// TwinCAT 3 PLC project MagnetSystem_PI4
// ProgramVersion: 3.1.4023.0
// libraries:
//   CanItfHelper, * (Beckhoff Automation LLC)
//   Tc2_Math, * (Beckhoff Automation GmbH)
//   Tc2_Standard, * (Beckhoff Automation GmbH)
//   Tc2_System, * (Beckhoff Automation GmbH)
//   Tc2_TcpIp, * (Beckhoff Automation GmbH)
//   Tc2_Utilities, * (Beckhoff Automation GmbH)
//   Tc3_Module, * (Beckhoff Automation GmbH)
//   Tc3_EventLogger,3.1.30.0,Beckhoff Automation GmbH
// project tree:
//   DUTs/ E_Command.TcDUT (not stored), E_MagState.TcDUT, E_Status.TcDUT, ST_Alarm_Base.TcDUT (not stored), ST_canRxdata.TcDUT (not stored), ST_Coil_Base.TcDUT (not stored), ST_Coil_Ext_Analog1.TcDUT (not stored), ST_Control.TcDUT (not stored), ST_EngVal.TcDUT (not stored), ST_InstFeedback.TcDUT (not stored), ST_RecipeLocal.TcDUT (not stored), ST_Setpoints.TcDUT (not stored), ST_PermissivesToMainPLC.TcDUT (not stored), ST_Recipe.TcDUT (not stored), ST_SysParameters.TcDUT, ST_Trip_Base.TcDUT (not stored), ST_UC_Status.TcDUT (not stored), ST_UC_Status_Dummy.TcDUT, ST_UCDevices.TcDUT, ST_UC_Trip_Base.TcDUT (not stored)
//   GVLs/ Alarms_DB.TcGVL (not stored), Command.TcGVL (not stored), Devices.TcGVL (not stored), HMI_DB.TcGVL, Input.TcGVL, GVL.TcGVL, InstrumentReading.TcGVL, IO.TcGVL (not stored), MCP_IO.TcGVL (not stored), Output.TcGVL (not stored), Permissives_DB.TcGVL (not stored), Recipe.TcGVL (not stored), Setpoints.TcGVL, Trips_DB.TcGVL, Tx_Config.TcGVL (not stored)
//   / PlcTask.TcTTO
//   POUs/ ADC_10V.TcPOU (not stored), ADC_5V.TcPOU (not stored), Alarms.TcPOU (not stored), Alarms_FB.TcPOU (not stored), Alias.TcPOU, AnalogConversion.TcPOU (not stored), Cal_ChargeTime.TcPOU, CanInterface.TcPOU (not stored), CAN_comm_old.TcPOU (not stored), CAN_comm.TcPOU (not stored), ChargeTimeCal.TcPOU (not stored), Delay2s.TcPOU (not stored), Graphs.TcPOU (not stored), Heartbeat.TcPOU (not stored), HMI.TcPOU (not stored), MAIN.TcPOU, MODE_SELECTION_1.TcPOU (not stored), Norm_x.TcPOU, Permissives.TcPOU (not stored), ChargeRlyClose_ChargerON_Seq.TcPOU (not stored), PWMO.TcPOU (not stored), Trips.TcPOU (not stored), Tx_MasterPLC.TcPOU, VoltageOutputCal.TcPOU (not stored)

CONFIGURATION MagnetSystem_PI4
    RESOURCE PLC ON TwinCAT3
        TASK PlcTask(INTERVAL := T#10ms, PRIORITY := 20);
        PROGRAM MAIN WITH PlcTask : MAIN;
    END_RESOURCE
END_CONFIGURATION

// ---- DUTs/E_MagState.TcDUT
{attribute 'qualified_only'}
{attribute 'strict'}
TYPE E_MagState :
(
	FULL_SHUTDOWN 	:= 0,
	IDLE			:= 1, 
	READY_TO_CHARGE := 2, 
	CHARGING		:= 3, 
	CHARGE_PAUSED	:= 4,
	READY_TO_SHOOT 	:= 5, 
	SHOOTING 		:= 6, 
	POST_SHOT 		:= 7, 
	//SHUTDOWN 		:= 8, //remove
	DUMPING			:= 9,
	TRIPPED			:= 10
);
END_TYPE

// ---- DUTs/E_Status.TcDUT
{attribute 'qualified_only'}
{attribute 'strict'}
{attribute 'to_string'}
TYPE E_Status :
(
	//Actual Magnetic State
	FULL_SHUTDOWN	:= 0,
	IDLE			:= 1, 
	READY_TO_CHARGE	:= 2, 
	CHARGING		:= 3, 
	CHARGING_PAUSED := 4,		
	READY_TO_SHOOT	:= 5, 
	SHOOTING		:= 6, 
	POST_SHOT		:= 7, 
	//SHUTDOWN		:= 8, 
	DUMPING			:= 9,
	TRIPPED			:= 10,
	MANUAL_MODE		:= 11 // LOCAL MODE
) ;
END_TYPE

// ---- DUTs/ST_SysParameters.TcDUT
TYPE ST_SysParameters :
STRUCT
	NumOfCaps				: INT := 2;
	Direction				: STRING[1] :='0';
	NumOfTurns				: INT := 0;
	DriverMapping			: STRING[10] := '0';
	MaxVoltagePerCap		: INT := 0;
	MaxVoltageTotal 		: INT := 0;
	CapacitancePerCap		: INT := 88;
	TotalCapacitance		: REAL := 0.0;
	TotalCircuitResistance	: REAL := 0.0;
	//TriggerTime				: INT := 0;
END_STRUCT
END_TYPE

// ---- DUTs/ST_UC_Status_Dummy.TcDUT
TYPE ST_UC_Status_Dummy EXTENDS ST_UC_Status :
STRUCT
	R2_06_UC_Rx_cobID : UDINT;
	R2_06_UC_Rx_data : ARRAY [0..7] OF BYTE;
END_STRUCT
END_TYPE

// ---- DUTs/ST_UCDevices.TcDUT
TYPE ST_UCDevices :
STRUCT
	Status : ST_UC_Status;
END_STRUCT
END_TYPE

// ---- GVLs/HMI_DB.TcGVL
{attribute 'qualified_only'}
VAR_GLOBAL
	chargePB			: BOOL;
	shootPB				: BOOL;
	dumpPB				: BOOL;
	StartPB				: BOOL;
	StopPB				: BOOL;
	PausePB				: BOOL;			 
	RemoteModeSelected	: BOOL;
	Idle_mode			: BOOL;
	SafetyOK			: BOOL;
	AllDumpRelaysOpen	: BOOL;
	AllACInterlocksClosed : BOOL;
	AllFlybackDiodesActive	: BOOL;
	IntrumentationFaulted	: BOOL;
	AllChargesAreActive		: BOOL;
	
	ReadyToChargeRunOutTime	: DINT := 0;
	ChargingRunOutTime		: DINT := 0;
	ChargePausedRunOutTime	: DINT := 0;
	ReadyToShootRunOutTime	: DINT := 0;				
	ShootingRunOutTime		: DINT := 0;
	PostShotRunOutTime		: DINT := 0;
	DumpingRunOutTime		: DINT := 0;
	
	CoilEnable				: ARRAY [1..10] OF BOOL;
	
END_VAR

// ---- GVLs/Input.TcGVL
{attribute 'qualified_only'}
VAR_GLOBAL
//***MCP
//EL1008 - DI
	R1_01_00 AT	%I*: BOOL; //Master stop PB not pressed - black pb on mcp
	R1_01_01 AT	%I*: BOOL; //case Estop circuit okay (Rly1 (120vac)
	R1_01_02 AT %I*: BOOL; //Automatic Mode Selected (NO)
	R1_01_03 AT %I*: BOOL; //24VDC OK
	R1_01_04 AT %I*: BOOL; //spare
	R1_01_05 AT %I*: BOOL; //spare
	R1_01_06 AT %I*: BOOL; //spare
	R1_01_07 AT %I*: BOOL; //spare


//***LCP
//EL3064 - AI
	R2_01_00 		AT %I*: INT;
	R2_01_00_Status AT %I*: WORD;
	
	R2_01_01		AT %I*: INT;
	R2_01_01_Status AT %I*: WORD;
	
	R2_01_02 		AT %I*: INT;
	R2_01_02_Status AT %I*: WORD;
	
//EL1008 - DI
	R2_03_00 AT %I*: BOOL;
	R2_03_01 AT %I*: BOOL;
	R2_03_02 AT %I*: BOOL;
	R2_03_03 AT %I*: BOOL;
	R2_03_04 AT %I*: BOOL;
	R2_03_05 AT %I*: BOOL;
	R2_03_06 AT %I*: BOOL;
	R2_03_07 AT %I*: BOOL;
	
	R2_04_00 AT %I*: BOOL;
	R2_04_01 AT %I*: BOOL;
	R2_04_02 AT %I*: BOOL;
	R2_04_03 AT %I*: BOOL;
	R2_04_04 AT %I*: BOOL;
	R2_04_05 AT %I*: BOOL; //spare
	R2_04_06 AT %I*: BOOL; //spare
	R2_04_07 AT %I*: BOOL; //spare

//EL6751 - CAN Open	
	
	//R2_06_UC_Rx AT %I*		: ARRAY [0..1] OF EXTCANQUEUE; // only used for raw address.
	// each Rack has 10 caps + 1 dummy varible to park the swapped cap
	R2_06_CapNumber AT %I* : ARRAY [1..10] OF  ST_UCDevices; //only used with DBC file.
	R2_06_UC_7F_status AT %I* : ST_UC_Status_Dummy;
	
//R3****** LCP2
//EL3064 - AI
	R3_01_00 		AT %I*: INT;
	R3_01_00_Status AT %I*: WORD;
	
	R3_01_01		AT %I*: INT;
	R3_01_01_Status AT %I*: WORD;
	
	R3_01_02 		AT %I*: INT;
	R3_01_02_Status AT %I*: WORD;
	
//EL1008 - DI
	R3_03_00 AT %I*: BOOL;
	R3_03_01 AT %I*: BOOL;
	R3_03_02 AT %I*: BOOL;
	R3_03_03 AT %I*: BOOL;
	R3_03_04 AT %I*: BOOL;
	R3_03_05 AT %I*: BOOL;
	R3_03_06 AT %I*: BOOL;
	R3_03_07 AT %I*: BOOL;
	
	R3_04_00 AT %I*: BOOL;
	R3_04_01 AT %I*: BOOL;
	R3_04_02 AT %I*: BOOL;
	R3_04_03 AT %I*: BOOL;
	R3_04_04 AT %I*: BOOL;
	R3_04_05 AT %I*: BOOL; //spare
	R3_04_06 AT %I*: BOOL; //rly - output relay
	R3_04_07 AT %I*: BOOL; //spare

//EL6751 - CAN Open	
	
	//R2_06_UC_Rx AT %I*		: ARRAY [0..1] OF EXTCANQUEUE; // only used for raw address.
	// each Rack has 10 caps + 1 dummy varible to park the swapped cap
	R3_06_CapNumber AT %I* : ARRAY [1..10] OF  ST_UCDevices; //only used with DBC file.
	R3_06_UC_7F_status AT %I* : ST_UC_Status_Dummy;
	//R3_06_UC_status AT %I* : ARRAY [1..10] OF ST_UC_Status;

	//R4 
	//R5	
	//..
	//R10

END_VAR

// ---- GVLs/GVL.TcGVL
{attribute 'qualified_only'}
VAR_GLOBAL
	
	//actual_magnet_systemState	: DINT;
	error_msg					: WORD;
	shot_going_OK				: BOOL;
	shot_is_done				: BOOL;
	//RequestedMagnetSysState		: DINT;
	cap_msg						: WORD; 
	
	test						: BOOL;
	ClearAllFaults				: BOOL;
	alarm_test					: BOOL;
	
	Analog_test					: REAL;
	
	fullshutdown_to_idle        : BOOL;
	idle_to_charge				: BOOL;
	idle_to_readyToCharge		: BOOL;
	readyToCharge_to_Charging	: BOOL;
	charge_to_pause				: BOOL;
	charge_to_readyToShoot		: BOOL;
	readyToShoot_to_Shoot		: BOOL;
	shoot_to_postShot			: BOOL;
	postShot_to_shutdown		: BOOL;
	shutdown_to_idle			: BOOL;
	dump_to_idle				: BOOL;
	
	AlwaysTrue					: BOOL;
	AlwaysFalse					: BOOL;
	
	AllSystemsDischarged		: BOOL;
	AllChargerReadywithSP		: BOOL;
END_VAR

// ---- GVLs/InstrumentReading.TcGVL
{attribute 'qualified_only'}
VAR_GLOBAL
	//LCP 1 Instrument reading
	R2_01_CH00 : REAL;
	R2_01_CH01 : REAL;
	R2_01_CH02 : REAL;
	
END_VAR

// ---- GVLs/Setpoints.TcGVL
{attribute 'qualified_only'}
VAR_GLOBAL
	//HMI Input -> Setpoints -> EngVal		-> PLC ---------> Tx_Config
	//						-> SysParameters-> PLC ---------> Tx_Config
	//										   PLC - Recipe -> Tx_Config 	 
	Coil : ARRAY[1..10] OF ST_Setpoints; // EngVal & SysParameters
	
END_VAR

// ---- GVLs/Trips_DB.TcGVL
{attribute 'qualified_only'}
VAR_GLOBAL
	Coil : ARRAY[1..10] OF ST_Trip_Base;
	
	AnyEstopPressed 			: BOOL;
	SystemTripped 				: BOOL;
	InstrumentationFaulted		: BOOL;
	AnyChargeRlyFail			: BOOL;
	AnyDumpRlyFail				: BOOL;
	AnyACInterlockFail			: BOOL;
	
	AnyDCPSU_fail				: BOOL;
	AnyHVisoRelayFailed			: BOOL;
	MachineTimedOut				: BOOL;
END_VAR

// ---- POUs/MAIN.TcPOU
PROGRAM MAIN
VAR
	
	status0:BOOL;
	
END_VAR

Alias();
CAN_comm();
Tx_MasterPLC();
AnalogConversion();
Permissives();
Trips();
MODE_SELECTION_1();
Alarms();
Heartbeat();
VoltageOutputCal();
Cal_ChargeTime();


//test
//IF MCP_IO.AutoModeSelected THEN
//	Output.R2_05_07 := heartbeat.pulse_1Hz;
//END_IF

	
//sample test
IF gvl.test = TRUE THEN
	Output.R2_05_00 := TRUE;
	ELSE 
		Output.R2_05_00 := FALSE; 	
END_IF;

END_PROGRAM

// ---- POUs/Alias.TcPOU
PROGRAM Alias
VAR
	i : INT := 1; //coil 1 - 10 
	j : INT := 1;  // msg 0-1 (could be 0-31 later)
END_VAR

//R1 = MCP**
//DI
	MCP_IO.MasterStopPB_Pressed					:= Input.R1_01_00;//NC
	//MCP_IO.MasterStopPB_Pressed					:= NOT Input.R2_04_07; //Temporarily used for testing.
	MCP_IO.CageEstopCircuitOK					:= Input.R1_01_01; //NO use R2_04_07 for dev test
	MCP_IO.RemoteModeSelected					:= Input.R1_01_02; // 0 = manual, 1=auto  *temporarily used for dev test
	MCP_IO.PSU1_DCOK							:= Input.R1_01_03;
	
//R2 = Coil 1
//AI
	Devices.Coil[1].ChargeVoltageFeedback_raw 	:= Input.R2_01_00;	
	Devices.Coil[1].CurrentFeedback_raw 		:= Input.R2_01_01;
	Devices.Coil[1].Measured_Bfield_raw 		:= Input.R2_01_02;
	
//PWM O
 	Output.R2_02_00 := Devices.Coil[1].ChargerSetpoint;
	Output.R2_02_01 := Devices.Coil[1].CurrentSetpoint;


//DI
	Devices.Coil[1].PSU0_active 				:= Input.R2_03_00;
	Devices.Coil[1].Local_StopPB_Pressed 		:= NOT Input.R2_03_01; //NC 
	Devices.Coil[1].DumpRelay1_closed 			:= Input.R2_03_02;
	Devices.Coil[1].DumpRelay2_closed 			:= Input.R2_03_03;
	//Devices.Coil[1].ChargeRelay_closed 			:= Input.R2_03_04;
	Devices.Coil[1].ChargerIsEnabled 			:= Input.R2_03_05;
	//Devices.Coil[1].FlybackD1_Alive 			:= Input.R2_03_06;
	//Devices.Coil[1].FlybackD2_Alive 			:= Input.R2_03_07;
	Devices.Coil[1].PSU1_DCOK					:= Input.R2_03_06;
	Devices.Coil[1].HVisolationRelayClosed		:= Input.R2_03_07; 
	
	Devices.Coil[1].DumpResistorTemperatureHigh := Input.R2_04_00;
	Devices.Coil[1].GroundLoopCurrentDetected 	:= Input.R2_04_01;
	Devices.Coil[1].CoilTemperatureHigh 		:= Input.R2_04_02;
	Devices.Coil[1].AC_Interlock_RlyClose		:= Input.R2_04_03;  //3P contactor
	Devices.Coil[1].LossPneumaticPressure       := Input.R2_04_04;
	//Spare Input.R2_04_05;  
	Devices.Coil[1].OutputRelayOpen				:= Input.R2_04_06; // rly 5
	//Spare Input.R2_04_07;  temp used for MCP estop input
	
//DQ
	Output.R2_05_00 := Devices.Coil[1].OpenDumpRelays;
	Output.R2_05_01 := Devices.Coil[1].closeChargeRelay;
	Output.R2_05_02 := Devices.Coil[1].enableOutputToCharger;
	Output.R2_05_03 := Devices.Coil[1].CloseACInterlockRly;  //3P contactor
	Output.R2_05_04 := Devices.Coil[1].CloseHVisolationRelay; // 24VDC to control 2 120Vac HV Ross Relayas  (rly6)
	Output.R2_05_05 := Devices.Coil[1].SystemFaulted; //LCP LED AMBER
	Output.R2_05_06 := Devices.Coil[1].SystemCharging;  //LCP LED RED (charging or Charged)
	Output.R2_05_07 := Devices.Coil[1].SystemReady;  // LCP LED GREEN
	
//CANOpen
	
	//Output.R2_05_CANrequest := CAN_comm.
	Output.R2_06_CANrequest.cobId := Devices.Coil[1].CanTx_config_ID;
	Output.R2_06_CANrequest.data[0] := Devices.Coil[1].CanTx_config_request[0];
	Output.R2_06_CANrequest.data[1] := Devices.Coil[1].CanTx_config_request[1];
	Output.R2_06_CANrequest.data[2] := Devices.Coil[1].CanTx_config_request[2];
	Output.R2_06_CANrequest.data[3] := Devices.Coil[1].CanTx_config_request[3];
	Output.R2_06_CANrequest.data[4] := Devices.Coil[1].CanTx_config_request[4];
	Output.R2_06_CANrequest.data[5] := Devices.Coil[1].CanTx_config_request[5];
	Output.R2_06_CANrequest.data[6] := Devices.Coil[1].CanTx_config_request[6];
	Output.R2_06_CANrequest.data[7] := Devices.Coil[1].CanTx_config_request[7];
	
	// input
FOR i := 1 TO 10 BY 1 DO
	FOR j := 1 TO 10 BY 1 DO 
		Devices.Coil[i].UltraCap[j].Elec_AveVolt 		:= Input.R2_06_CapNumber[j].Status.Elec_AveVolt; //per cell
		Devices.Coil[i].UltraCap[j].Elec_Balancing 		:= Input.R2_06_CapNumber[j].Status.Elec_Balancing; // 0x0[Not Active], 0x1[Active], 0x2[Error], 0x3[Not Available]
		Devices.Coil[i].UltraCap[j].Elec_HighestVolt 	:= Input.R2_06_CapNumber[j].Status.Elec_HighestVolt; //per cell
		Devices.Coil[i].UltraCap[j].Elec_Imbalance 		:= Input.R2_06_CapNumber[j].Status.Elec_Imbalance;  // 0x0[No Warnings], 0x1[Warning Active], 0x2[Alarm Active], 0x3[Not Available]
		Devices.Coil[i].UltraCap[j].Elec_OverVoltage	:= Input.R2_06_CapNumber[j].Status.Elec_OverVoltage;  // 0x0[No Warnings], 0x1[Warning Active], 0x2[Alarm Active], 0x3[NOT Available] 
		Devices.Coil[i].UltraCap[j].Elec_VoltageSum		:= Input.R2_06_CapNumber[j].Status.Elec_VoltageSum; //total voltage in one UC
		Devices.Coil[i].UltraCap[j].Therm_HighestCell	:= Input.R2_06_CapNumber[j].Status.Therm_HighestCell; //C
		Devices.Coil[i].UltraCap[j].Therm_HighTemp		:= Input.R2_06_CapNumber[j].Status.Therm_HighTemp;  //0x0[No Warnings], 0x1[Warning Active], 0x2[Alarm Active], 0x3[NOT Available]
	END_FOR;
END_FOR;
	Devices.Coil[1].UltraCap_Dummy.R2_06_UC_Rx_cobID := Input.R2_06_UC_7F_status.R2_06_UC_Rx_cobID;
	Devices.Coil[1].UltraCap_Dummy.R2_06_UC_Rx_data := Input.R2_06_UC_7F_status.R2_06_UC_Rx_data;

//Recipe: Coil enable from screenroom
IF MCP_IO.RemoteModeSelected = TRUE OR HMI_DB.RemoteModeSelected = TRUE THEN
	FOR i := 1 TO 10 BY 1 DO
		Devices.Coil[i].CoilEnabled :=  Recipe.Coil[i].CoilEnable;
	END_FOR;
	
ELSIF MCP_IO.RemoteModeSelected = FALSE OR HMI_DB.RemoteModeSelected = FALSE THEN
	FOR i := 1 TO 10 BY 1 DO
		Devices.Coil[i].CoilEnabled :=  HMI_DB.CoilEnable[i];	
	END_FOR;
END_IF;


IF i > 10 THEN
	i := 1;
END_IF;

IF j > 10 THEN
	j := 1;
END_IF;

END_PROGRAM

// ---- POUs/Tx_MasterPLC.TcPOU
PROGRAM Tx_MasterPLC
VAR
	i : INT := 1;
	j : INT := 1;
	TotalCapacitance_REAL : ARRAY[1..10] OF REAL;
	
END_VAR

//Calculations for Max Total Voltage and Total Capacitance
FOR i := 1 TO 10 BY 1 DO
	Setpoints.Coil[i].SysParameters.MaxVoltageTotal := Setpoints.Coil[i].SysParameters.NumOfCaps * Setpoints.Coil[i].SysParameters.MaxVoltagePerCap;
	TotalCapacitance_REAL[i] := INT_TO_REAL(Setpoints.Coil[i].SysParameters.CapacitancePerCap) / INT_TO_REAL(Setpoints.Coil[i].SysParameters.NumOfCaps);
	Setpoints.Coil[i].SysParameters.TotalCapacitance := TotalCapacitance_REAL[i];
END_FOR


//Grouping systemParameters and configuration for sending to main plc
FOR i := 1 TO 10 BY 1 DO
	Tx_Config.CoilSP[i].SysParameters.Direction := Setpoints.Coil[i].SysParameters.Direction;
	Tx_Config.CoilSP[i].SysParameters.NumOfTurns := Setpoints.Coil[i].SysParameters.NumOfTurns;
	Tx_Config.CoilSP[i].SysParameters.DriverMapping := Setpoints.Coil[i].SysParameters.DriverMapping;
	Tx_Config.CoilSP[i].SysParameters.NumOfCaps := Setpoints.Coil[i].SysParameters.NumOfCaps;
	Tx_Config.CoilSP[i].SysParameters.MaxVoltagePerCap := Setpoints.Coil[i].SysParameters.MaxVoltagePerCap;
	Tx_Config.CoilSP[i].SysParameters.MaxVoltageTotal := Setpoints.Coil[i].SysParameters.MaxVoltageTotal;
	Tx_Config.CoilSP[i].SysParameters.CapacitancePerCap := Setpoints.Coil[i].SysParameters.CapacitancePerCap;
	Tx_Config.CoilSP[i].SysParameters.TotalCapacitance := Setpoints.Coil[i].SysParameters.TotalCapacitance;
	Tx_Config.CoilSP[i].SysParameters.TotalCircuitResistance := Setpoints.Coil[i].SysParameters.TotalCircuitResistance;
	
	Tx_Config.CoilSP[i].RecipeLocal.chargerSetpoint	:= Setpoints.Coil[i].RecipeLocal.chargerSetpoint;//calculated locally, thought the mainPLC might want to have this 
	Tx_Config.CoilSP[i].Recipe.CoilEnable			:= Recipe.Coil[i].CoilEnable;
	Tx_Config.CoilSP[i].Recipe.CurrentDuration	:= Recipe.Coil[i].CurrentDuration; //total charge time?
	Tx_Config.CoilSP[i].Recipe.currentSetpoint	:= Recipe.Coil[i].currentSetpoint;
	Tx_Config.CoilSP[i].Recipe.TriggerTime		:= Recipe.Coil[i].TriggerTime;
	
	Tx_Config.CoilInst[i].ChargerVolt := Devices.Coil[i].ChargeVoltageFeedback;
	
	FOR j := 1 TO 15 BY 1 DO 
		Tx_Config.CoilInst[i].CapVolt[j] := INT_TO_REAL (Devices.Coil[i].CapVoltage[j]); //1-15 uc
		Tx_Config.CoilInst[i].TotalVoltage := Devices.Coil[i].TotalVoltage;
	END_FOR
	
	Tx_Config.CoilInst[i].Cur := Devices.Coil[i].CurrentFeedback;
	
END_FOR

//run out time of each state
Tx_Config.ReadyToChargeRunOutTime := TIME_TO_REAL (MODE_SELECTION_1.ReadyToChargeRunOutTMR_PT);
Tx_Config.ChargingRunOutTime := TIME_TO_REAL (MODE_SELECTION_1.ChargingRunOutTMR_PT);
Tx_Config.ChargePausedRunOutTime := TIME_TO_REAL (MODE_SELECTION_1.ChargePausedRunOutTMR_PT);
Tx_Config.ReadyToShootRunOutTime := TIME_TO_REAL (MODE_SELECTION_1.ReadyToShootRunOutTMR_PT);
Tx_Config.ShootingRunOutTime := TIME_TO_REAL (MODE_SELECTION_1.ShootingRunOutTMR_PT);
Tx_Config.PostShotRunOutTime := TIME_TO_REAL (MODE_SELECTION_1.PostShotRunOutTMR_PT);
Tx_Config.DumpingRunOutTime := TIME_TO_REAL (MODE_SELECTION_1.DumpingRunOutTMR_PT);

//voltage and current feedback???

//TxRx
(*
FB_ReadAdsSymByName (
			bRead		:= TRUE, // on or off
			sNetID		:= 5.104.224.86.1.333, //AmsNetID
			nPort		:= 852, // plc port
			sVarName	:= E_Command,  //read from
			nDestAddr	:= E_Command, //write to 
			nLen		:= 2, //2 bytes	
			);

FB_WriteAdsSymByName (
			bWrite		:= TRUE,
			sNetID		:= 5.1.121.21.21.2,
			nPort		:= 851,
			sVarName	:= E_Status,
			nSrcAddr	:= E_Status,
			nLen		:= 2, //2byte
			);
*)


IF i > 10 THEN 
	i := 1;
END_IF

IF j > 15 THEN 
	j := 1;
END_IF

END_PROGRAM

// ---- POUs/Cal_ChargeTime.TcPOU
PROGRAM Cal_ChargeTime
VAR
	chargetimeCal : ARRAY [1..10] OF ChargeTimeCal;
	Tuntilfullycharged : ARRAY [1..10] OF REAL;
	i : INT := 1;
END_VAR


FOR i := 1 TO 10 BY 1 DO
	chargetimeCal[i] (I_setpoint := setpoints.Coil[i].Recipe.currentSetpoint, 
					t_duration := setpoints.Coil[i].Recipe.CurrentDuration, 
					NumOfCaps := setpoints.Coil[i].SysParameters.NumOfCaps,
					C_percap := setpoints.Coil[i].SysParameters.CapacitancePerCap,
					VMAXperCap := setpoints.Coil[i].SysParameters.MaxVoltagePerCap,
					R_coil := setpoints.Coil[i].SysParameters.TotalCircuitResistance,
					L_coil := 0.5,
					VMAXcharger := 1500,
					Pcharger := 15000,
					NumOfCharger := 4);
				
Tuntilfullycharged[i] := chargetimeCal[i].Tuntilfullcharge;
END_FOR;

IF i > 10 THEN 
	i := 1;
END_IF

END_PROGRAM

// ---- POUs/Norm_x.TcPOU
FUNCTION Norm_x : REAL
VAR_INPUT
	raw_input : REAL;
	x_max : REAL := 32767;
	x_min : REAL := 0;
END_VAR
VAR
END_VAR

// 0 - 10V AI INPUT 
Norm_x := (raw_input - x_min) / (x_max - x_min);

END_FUNCTION
